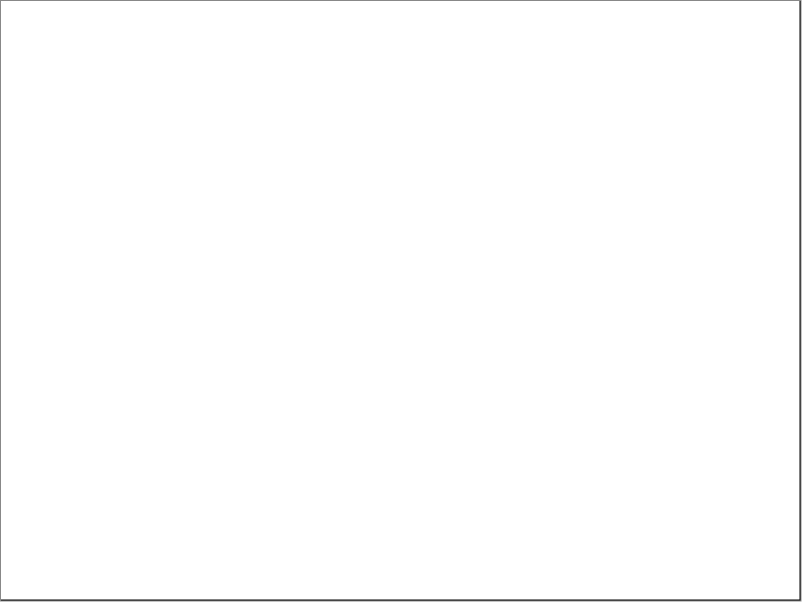
VISUALIZATION F00_Blank  // 802x602
    Rectangle (0,0 800x600)
END_VISUALIZATION

(* stored: Version 1.1.0.1, ProductVersion 3.1.4022.7
   Visu F00_Blank: Id {ca756281-9453-48c0-b4fe-67467ed98ee3} *)
